(* CODESYS project CintasSoplado.project
   Title: CintasSoplado
   Version: 0.0.0.0
   Author: serbogr1

Project tree, tasks and I/O mapping:
  MyController : TM241CE40R, Schneider Electric, order no. TM241CE40R, version 4.0.6.18
    application Application
      libraries: Toolbox, 2.2.0.0 (Schneider Electric); VisuDialogs, * (System)
      task MAST (cyclic, interval 50 ms, priority 15) calls ProcesoUno, ProcesoDos, Pulsadores, PID, Gestion_HMI, Control_HMI, Soplado_AUT, Operaciones_MAT
      global variables GVL
      visualisation Control_HMIW
      image pool ImagePool
      program ProcesoDos [SFC]: E2_active, E10_active
      program PID [LD]
      program ProcesoUno [SFC]: E8_active, E7_active, E9_active, E10_active, E11_active, E12_active, E1_active
      program Pulsadores [LD]
      program Gestion_HMI [LD]
      program Control_HMI [ST]
      program Operaciones_MAT [ST]
      program Soplado_AUT [SFC]: E1_active, E3_active, E2_active, E4_active, E5_active, E6_active, E7_active
    DI : Digital Inputs, Schneider Electric, version 4.0.6.18
        input  idwDI_IDW0 : DWORD  // IDW0
        input  ibDI_IB1 : BYTE  // IB1
    DQ : Digital Outputs, Schneider Electric, version 4.0.6.18
        output qwDQ_QW0 : WORD  // QW0
        output qbDQ_QB1 : BYTE  // QB1
    Counters : Counters, Schneider Electric, version 4.0.6.18
    Pulse_Generators : Pulse Generators, Schneider Electric, version 4.0.6.18
    Cartridge_1 : Cartridge, Schneider Electric, version 4.0.6.18
      TMC4AI2 : TMC4AI2, Schneider Electric, order no. TMC4AI2, version 1.0.1.0
          input  iiTMC4AI2_IW0 : INT  // IW0
          input  iiTMC4AI2_IW1 : INT  // IW1
          input  ibTMC4AI2_IW2 : BYTE  // IW2
    Cartridge_2 : Cartridge, Schneider Electric, version 4.0.6.18
      TMC4AQ2 : TMC4AQ2, Schneider Electric, order no. TMC4AQ2, version 1.0.1.1
          output qiTMC4AQ2_QW0 : INT  // QW0
          output qiTMC4AQ2_QW1 : INT  // QW1
          input  ibTMC4AQ2_IW0 : BYTE  // IW0
    IO_Bus : IO bus - TM3, Schneider Electric, version 4.0.6.18
    COM_Bus : COM bus, Schneider Electric, version 4.0.6.18
    Ethernet_1 : Ethernet Network, Schneider Electric, version 4.0.6.18
        settings: WebServer = TRUE; FTP Server = TRUE; SoMachine Protocol = TRUE; Modbus Server = TRUE; NetManage Protocol = TRUE; SNMP protocol = TRUE; Enable Routing = FALSE; WebVisu protocol = TRUE; DHCP Server Active = FALSE
    Serial_Line_1 : Serial line, Schneider Electric, version 4.0.6.18
      SoMachine_Network_Manager : SoMachine-Network Manager, Schneider Electric, version 4.0.0.2
    Serial_Line_2 : Serial line, Schneider Electric, version 4.0.6.18
      Modbus_Manager : Modbus Manager, Schneider Electric, version 4.0.0.2
  text list GlobalTextList
*)

// MyController/Application/GVL
VAR_GLOBAL
	iTiempoFresado      AT %MW100: INT :=2;	
	iTiempoTaladrado    AT %MW101: INT :=2;
	iTiempoSoplado      AT %MW102: INT :=2;
	rReferencia         AT %MD118: REAL:=-0.75;
	iPosInicioGrados    AT %MD105: REAL:=0;
	iPosSopladoGrados   AT %MD106: REAL:=20;
    iPosSopladoReposo	AT %MD99 : REAL:=-37;
	iGradosAguja        AT %MW104: INT;
	rPosicionActual              : REAL;	
END_VAR

// MyController/Application/ProcesoUno
PROGRAM ProcesoUno
VAR
	bS_FC_Empujador_1          AT %IX0.0: BOOL; (*I1*)
	bS_IC_Empujador_1          AT %IX0.1: BOOL; (*I2*)
	bS_FC_Empujador_2          AT %IX0.2: BOOL; (*I3*)
	bS_IC_Empujador_2          AT %IX0.3: BOOL; (*I4*)
	bS_FT_Empujador_1          AT %IX0.4: BOOL; (*I5*)
	bS_FT_Fresadora            AT %IX0.5: BOOL; (*I6*)
	bS_FT_Carga                AT %IX0.6: BOOL; (*I7*)
	bS_FT_Taladro              AT %IX0.7: BOOL; (*I8*)
	bS_FT_Salida               AT %IX1.0: BOOL; (*I9*)

    bSiguientePieza            AT %MX0.4: BOOL; (*Activa cuando se puede poner la siguiente pieza*)
	FalloSensores              AT %MX0.5: BOOL:=FALSE;	
	CintaFresadoraP1                    : BOOL;	
	CintaTaladroP1                      : BOOL;	
	CintaAlimentacionP1                 : BOOL;
	MotorFresadora                      : BOOL;
END_VAR

VAR_OUTPUT
	tEmpujador_1   : TIME:=T#1S;
	tFresado       : TIME:=T#1S;
END_VAR

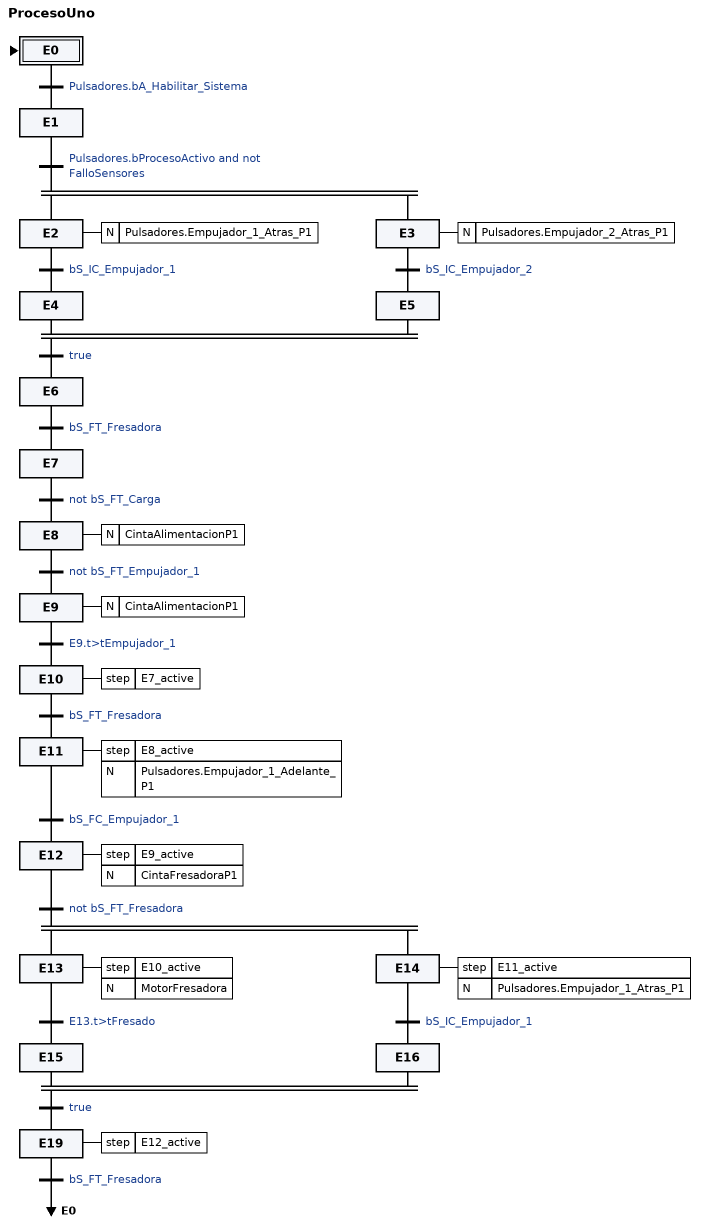
INITIAL_STEP E0:
END_STEP
TRANSITION FROM E0 TO E1
    := Pulsadores.bA_Habilitar_Sistema;
END_TRANSITION
STEP E1:
END_STEP
TRANSITION FROM E1 TO (E2, E3)
    := Pulsadores.bProcesoActivo and not FalloSensores;
END_TRANSITION
STEP E2:
    Pulsadores.Empujador_1_Atras_P1(N);
END_STEP
TRANSITION FROM E2 TO E4
    := bS_IC_Empujador_1;
END_TRANSITION
STEP E4:
END_STEP
STEP E3:
    Pulsadores.Empujador_2_Atras_P1(N);
END_STEP
TRANSITION FROM E3 TO E5
    := bS_IC_Empujador_2;
END_TRANSITION
STEP E5:
END_STEP
TRANSITION FROM (E4, E5) TO E6
    := true;
END_TRANSITION
STEP E6:
END_STEP
TRANSITION FROM E6 TO E7
    := bS_FT_Fresadora;
END_TRANSITION
STEP E7:
END_STEP
TRANSITION FROM E7 TO E8
    := not bS_FT_Carga;
END_TRANSITION
STEP E8:
    CintaAlimentacionP1(N);
END_STEP
TRANSITION FROM E8 TO E9
    := not bS_FT_Empujador_1;
END_TRANSITION
STEP E9:
    CintaAlimentacionP1(N);
END_STEP
TRANSITION FROM E9 TO E10
    := E9.t>tEmpujador_1;
END_TRANSITION
STEP E10:
    E7_active(N);  // step action
END_STEP
TRANSITION FROM E10 TO E11
    := bS_FT_Fresadora;
END_TRANSITION
STEP E11:
    E8_active(N);  // step action
    Pulsadores.Empujador_1_Adelante_P1(N);
END_STEP
TRANSITION FROM E11 TO E12
    := bS_FC_Empujador_1;
END_TRANSITION
STEP E12:
    E9_active(N);  // step action
    CintaFresadoraP1(N);
END_STEP
TRANSITION FROM E12 TO (E13, E14)
    := not bS_FT_Fresadora;
END_TRANSITION
STEP E13:
    E10_active(N);  // step action
    MotorFresadora(N);
END_STEP
TRANSITION FROM E13 TO E15
    := E13.t>tFresado;
END_TRANSITION
STEP E15:
END_STEP
STEP E14:
    E11_active(N);  // step action
    Pulsadores.Empujador_1_Atras_P1(N);
END_STEP
TRANSITION FROM E14 TO E16
    := bS_IC_Empujador_1;
END_TRANSITION
STEP E16:
END_STEP
TRANSITION FROM (E15, E16) TO E19
    := true;
END_TRANSITION
STEP E19:
    E12_active(N);  // step action
END_STEP
TRANSITION FROM E19 TO E0
    := bS_FT_Fresadora;
END_TRANSITION

ACTION E8_active:
IF bS_FT_Carga THEN
	bSiguientePieza := TRUE;
ELSIF NOT bS_FT_Carga THEN
	bSiguientePieza := FALSE;
END_IF
END_ACTION

ACTION E7_active:
IF bS_FT_Carga THEN
	bSiguientePieza := TRUE;
ELSIF NOT bS_FT_Carga THEN
	bSiguientePieza := FALSE;
END_IF
END_ACTION

ACTION E9_active:
IF bS_FT_Carga THEN
	bSiguientePieza := TRUE;
ELSIF NOT bS_FT_Carga THEN
	bSiguientePieza := FALSE;
END_IF
END_ACTION

ACTION E10_active:
IF bS_FT_Carga THEN
	bSiguientePieza := TRUE;
ELSIF NOT bS_FT_Carga THEN
	bSiguientePieza := FALSE;
END_IF

	tFresado := INT_TO_TIME(iTiempoFresado*1000);
END_ACTION

ACTION E11_active:
IF bS_FT_Carga THEN
	bSiguientePieza := TRUE;
ELSIF NOT bS_FT_Carga THEN
	bSiguientePieza := FALSE;
END_IF
END_ACTION

ACTION E12_active:
IF bS_FT_Carga THEN
	bSiguientePieza := TRUE;
ELSIF NOT bS_FT_Carga THEN
	bSiguientePieza := FALSE;
END_IF
END_ACTION

ACTION E1_active:
IF NOT Pulsadores.bBotonInicioHMIS THEN
	IF NOT bS_FT_Carga THEN
		FalloSensores:=TRUE;	
	END_IF
	IF NOT bS_FT_Empujador_1 THEN
		FalloSensores:=TRUE;
	END_IF
	IF NOT bS_FT_Fresadora THEN
		FalloSensores:=TRUE;
	END_IF
	IF NOT bS_FT_Taladro THEN
		FalloSensores:=TRUE;
	END_IF
	IF NOT bS_FT_Salida THEN
		FalloSensores:=TRUE;	
	END_IF
	
	IF bS_FT_Carga AND bS_FT_Empujador_1 AND bS_FT_Fresadora AND bS_FT_Taladro AND bS_FT_Salida THEN
		FalloSensores:=FALSE;			
	END_IF
END_IF
END_ACTION

END_PROGRAM

// MyController/Application/Pulsadores
PROGRAM Pulsadores
VAR
	bA_M_Empujador_1_Adelante  AT %QX0.4: BOOL; (*Q1*)
	bA_M_Empujador_1_Atras     AT %QX0.5: BOOL; (*Q2*)
	bA_M_Empujador_2_Adelante  AT %QX0.6: BOOL; (*Q3*)
	bA_M_Empujador_2_Atras     AT %QX0.7: BOOL; (*Q4*)	
	bA_M_Cinta_Alimentacion    AT %QX1.0: BOOL; (*Q5*)	
	bA_M_Cinta_Fresadora       AT %QX1.1: BOOL; (*Q6*)
	bA_M_Fresadora             AT %QX1.2: BOOL; (*Q7*)	
	bA_M_Cinta_Taladro         AT %QX1.3: BOOL; (*Q8*)	
	bA_M_Taladro               AT %QX1.4: BOOL; (*Q9*)	
	bA_M_Cinta_Salida          AT %QX1.5: BOOL; (*Q10*)		
	bA_Habilitar_Sistema       AT %QX1.6: BOOL; (*Q11*)	
	
	bBotonEmergenciaHMIS       AT %MX0.0: BOOL; (*Boton Emergencia HMI y HMIW*)	
	bBotonEncendidoHMIS        AT %MX0.1: BOOL; (*Boton Encendido HMI y HMIW*)	
	bBotonInicioHMIS           AT %MX0.2: BOOL; (*Boton Inicio HMI y HMIW*)	
	bAlarma_ON                 AT %MX0.3: BOOL; (*Activa cuando se pulsa alarma*)
	bProcesoActivo                      : BOOL; (*Activa cuando se pulsa inicio*)	
	
	Empujador_1_Adelante_P1             : BOOL;
	Empujador_1_Adelante_P2             : BOOL;
	Empujador_2_Adelante_P1             : BOOL;	
    Empujador_2_Adelante_P2             : BOOL;
	Empujador_1_Atras_P1                : BOOL;
	Empujador_1_Atras_P2                : BOOL;	
	Empujador_2_Atras_P1                : BOOL;
	Empujador_2_Atras_P2                : BOOL;	
	bStopSoplado                        : BOOL;	
	rLongTime                           : INT;
END_VAR

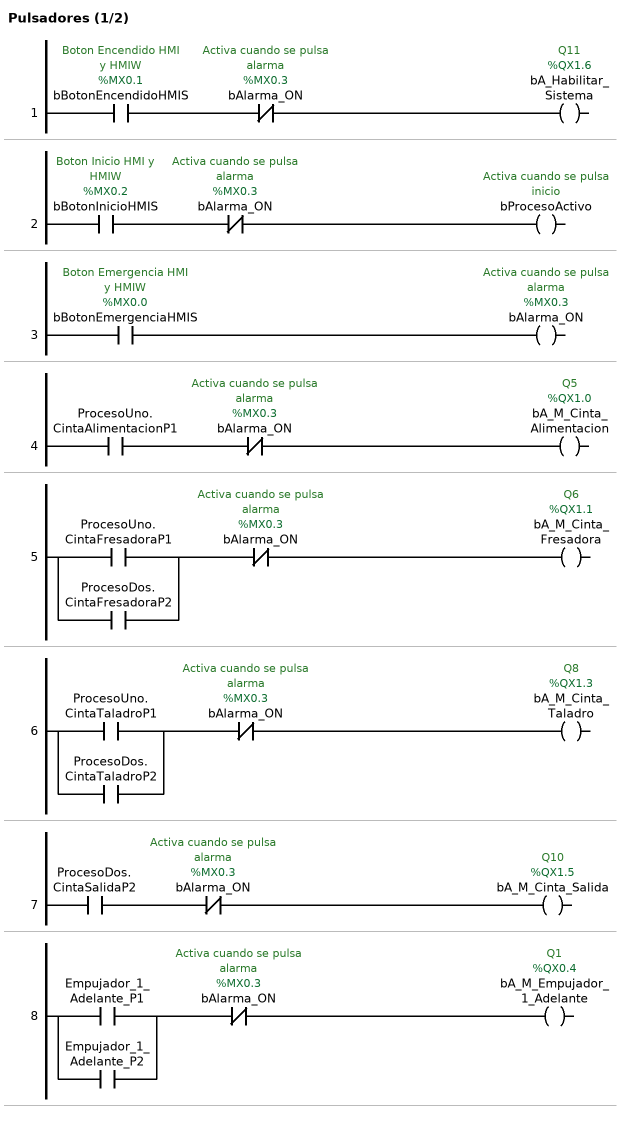
// NETWORK 1
//   bBotonEncendidoHMIS: Boton Encendido HMI y HMIW | AT %MX0.1
//   bAlarma_ON: Activa cuando se pulsa alarma | AT %MX0.3
//   bA_Habilitar_Sistema: Q11 | AT %QX1.6
bA_Habilitar_Sistema := bBotonEncendidoHMIS AND NOT bAlarma_ON;

// NETWORK 2
//   bBotonInicioHMIS: Boton Inicio HMI y HMIW | AT %MX0.2
//   bAlarma_ON: Activa cuando se pulsa alarma | AT %MX0.3
//   bProcesoActivo: Activa cuando se pulsa inicio
bProcesoActivo := bBotonInicioHMIS AND NOT bAlarma_ON;

// NETWORK 3
//   bBotonEmergenciaHMIS: Boton Emergencia HMI y HMIW | AT %MX0.0
//   bAlarma_ON: Activa cuando se pulsa alarma | AT %MX0.3
bAlarma_ON := bBotonEmergenciaHMIS;

// NETWORK 4
//   bAlarma_ON: Activa cuando se pulsa alarma | AT %MX0.3
//   bA_M_Cinta_Alimentacion: Q5 | AT %QX1.0
bA_M_Cinta_Alimentacion := ProcesoUno.CintaAlimentacionP1 AND NOT bAlarma_ON;

// NETWORK 5
//   bAlarma_ON: Activa cuando se pulsa alarma | AT %MX0.3
//   bA_M_Cinta_Fresadora: Q6 | AT %QX1.1
bA_M_Cinta_Fresadora := (ProcesoUno.CintaFresadoraP1 OR ProcesoDos.CintaFresadoraP2) AND NOT bAlarma_ON;

// NETWORK 6
//   bAlarma_ON: Activa cuando se pulsa alarma | AT %MX0.3
//   bA_M_Cinta_Taladro: Q8 | AT %QX1.3
bA_M_Cinta_Taladro := (ProcesoUno.CintaTaladroP1 OR ProcesoDos.CintaTaladroP2) AND NOT bAlarma_ON;

// NETWORK 7
//   bAlarma_ON: Activa cuando se pulsa alarma | AT %MX0.3
//   bA_M_Cinta_Salida: Q10 | AT %QX1.5
bA_M_Cinta_Salida := ProcesoDos.CintaSalidaP2 AND NOT bAlarma_ON;

// NETWORK 8
//   bAlarma_ON: Activa cuando se pulsa alarma | AT %MX0.3
//   bA_M_Empujador_1_Adelante: Q1 | AT %QX0.4
bA_M_Empujador_1_Adelante := (Empujador_1_Adelante_P1 OR Empujador_1_Adelante_P2) AND NOT bAlarma_ON;

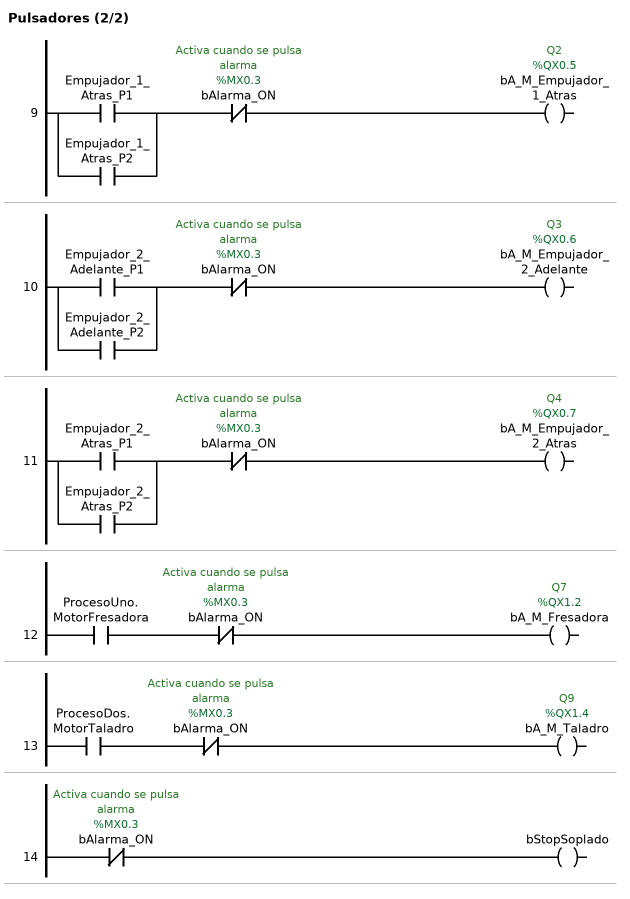
// NETWORK 9
//   bAlarma_ON: Activa cuando se pulsa alarma | AT %MX0.3
//   bA_M_Empujador_1_Atras: Q2 | AT %QX0.5
bA_M_Empujador_1_Atras := (Empujador_1_Atras_P1 OR Empujador_1_Atras_P2) AND NOT bAlarma_ON;

// NETWORK 10
//   bAlarma_ON: Activa cuando se pulsa alarma | AT %MX0.3
//   bA_M_Empujador_2_Adelante: Q3 | AT %QX0.6
bA_M_Empujador_2_Adelante := (Empujador_2_Adelante_P1 OR Empujador_2_Adelante_P2) AND NOT bAlarma_ON;

// NETWORK 11
//   bAlarma_ON: Activa cuando se pulsa alarma | AT %MX0.3
//   bA_M_Empujador_2_Atras: Q4 | AT %QX0.7
bA_M_Empujador_2_Atras := (Empujador_2_Atras_P1 OR Empujador_2_Atras_P2) AND NOT bAlarma_ON;

// NETWORK 12
//   bAlarma_ON: Activa cuando se pulsa alarma | AT %MX0.3
//   bA_M_Fresadora: Q7 | AT %QX1.2
bA_M_Fresadora := ProcesoUno.MotorFresadora AND NOT bAlarma_ON;

// NETWORK 13
//   bAlarma_ON: Activa cuando se pulsa alarma | AT %MX0.3
//   bA_M_Taladro: Q9 | AT %QX1.4
bA_M_Taladro := ProcesoDos.MotorTaladro AND NOT bAlarma_ON;

// NETWORK 14
//   bAlarma_ON: Activa cuando se pulsa alarma | AT %MX0.3
bStopSoplado := NOT bAlarma_ON;

END_PROGRAM

// MyController/Application/ProcesoDos
PROGRAM ProcesoDos
VAR	
    CintaSalidaP2                 : BOOL;
    MotorTaladro                  : BOOL;
	CintaFresadoraP2              : BOOL;
	CintaTaladroP2                : BOOL;	

	rPiezasTerminadas   AT %MW103 : INT:=0;		
	tTaladrado                    : TIME:=T#2S;
	tEmpujador_2                  : TIME:=T#2S;	
END_VAR

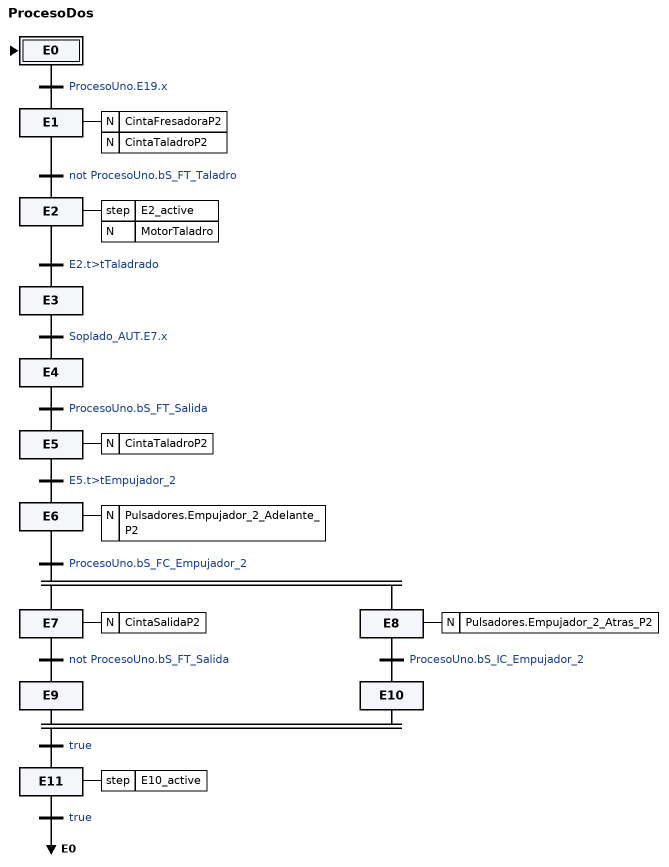
INITIAL_STEP E0:
END_STEP
TRANSITION FROM E0 TO E1
    := ProcesoUno.E19.x;
END_TRANSITION
STEP E1:
    CintaFresadoraP2(N);
    CintaTaladroP2(N);
END_STEP
TRANSITION FROM E1 TO E2
    := not ProcesoUno.bS_FT_Taladro;
END_TRANSITION
STEP E2:
    E2_active(N);  // step action
    MotorTaladro(N);
END_STEP
TRANSITION FROM E2 TO E3
    := E2.t>tTaladrado;
END_TRANSITION
STEP E3:
END_STEP
TRANSITION FROM E3 TO E4
    := Soplado_AUT.E7.x;
END_TRANSITION
STEP E4:
END_STEP
TRANSITION FROM E4 TO E5
    := ProcesoUno.bS_FT_Salida;
END_TRANSITION
STEP E5:
    CintaTaladroP2(N);
END_STEP
TRANSITION FROM E5 TO E6
    := E5.t>tEmpujador_2;
END_TRANSITION
STEP E6:
    Pulsadores.Empujador_2_Adelante_P2(N);
END_STEP
TRANSITION FROM E6 TO (E7, E8)
    := ProcesoUno.bS_FC_Empujador_2;
END_TRANSITION
STEP E7:
    CintaSalidaP2(N);
END_STEP
TRANSITION FROM E7 TO E9
    := not ProcesoUno.bS_FT_Salida;
END_TRANSITION
STEP E9:
END_STEP
STEP E8:
    Pulsadores.Empujador_2_Atras_P2(N);
END_STEP
TRANSITION FROM E8 TO E10
    := ProcesoUno.bS_IC_Empujador_2;
END_TRANSITION
STEP E10:
END_STEP
TRANSITION FROM (E9, E10) TO E11
    := true;
END_TRANSITION
STEP E11:
    E10_active(N);  // step action
END_STEP
TRANSITION FROM E11 TO E0
    := true;
END_TRANSITION

ACTION E2_active:
  
IF Gestion_HMI.bSum_T_Taladrado THEN
	iTiempoTaladrado := iTiempoTaladrado + 1;
END_IF
IF Gestion_HMI.bRes_T_Taladrado THEN
	iTiempoTaladrado := iTiempoTaladrado - 1;
END_IF

	tTaladrado := INT_TO_TIME(iTiempoTaladrado*1000);
END_ACTION

ACTION E10_active:
IF NOT ProcesoUno.bS_FT_Salida THEN
	rPiezasTerminadas := rPiezasTerminadas + 1;
END_IF
END_ACTION

END_PROGRAM

// MyController/Application/Gestion_HMI
PROGRAM Gestion_HMI
VAR
	bRes_T_Fresado              AT %MX1.0: BOOL;
	bSum_T_Fresado              AT %MX1.1: BOOL;
	bRes_T_Taladrado            AT %MX1.2: BOOL;
	bSum_T_Taladrado            AT %MX1.3: BOOL;
	bRes_T_Soplado              AT %MX1.4: BOOL;
	bSum_T_Soplado              AT %MX1.5: BOOL;		
	bRes_AnguloInicio           AT %MX1.6: BOOL;		
	bSum_AnguloInicio           AT %MX1.7: BOOL;
	bRes_AnguloSoplado          AT %MX2.0: BOOL;
	bSum_AnguloSoplado          AT %MX2.1: BOOL;	

	bSe_FT_Carga                AT %MX2.2: BOOL; 
	bSe_FT_Empujador_1          AT %MX2.3: BOOL; 
	bSe_FC_Empujador_1          AT %MX2.4: BOOL;
	bSe_FT_Fresadora            AT %MX2.5: BOOL; 	
	bSe_FT_Taladro              AT %MX2.6: BOOL;
	bSe_FC_Empujador_2          AT %MX2.7: BOOL;  
	bSe_FT_Salida               AT %MX3.0: BOOL; 
	bAe_M_Empujador_1_Adelante  AT %MX3.1: BOOL;
	bAe_M_Fresadora             AT %MX3.2: BOOL;
	bAe_M_Taladro               AT %MX3.3: BOOL;
	bAe_M_Empujador_2_Adelante  AT %MX3.4: BOOL;	

END_VAR

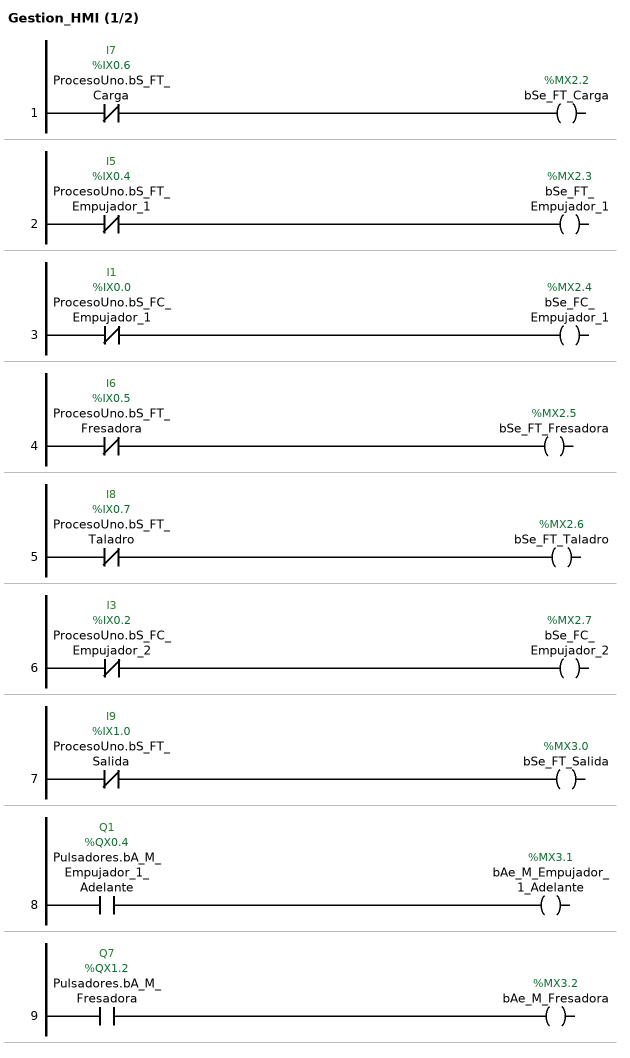
// NETWORK 1
//   ProcesoUno.bS_FT_Carga: I7 | AT %IX0.6
//   bSe_FT_Carga: AT %MX2.2
bSe_FT_Carga := NOT ProcesoUno.bS_FT_Carga;

// NETWORK 2
//   ProcesoUno.bS_FT_Empujador_1: I5 | AT %IX0.4
//   bSe_FT_Empujador_1: AT %MX2.3
bSe_FT_Empujador_1 := NOT ProcesoUno.bS_FT_Empujador_1;

// NETWORK 3
//   ProcesoUno.bS_FC_Empujador_1: I1 | AT %IX0.0
//   bSe_FC_Empujador_1: AT %MX2.4
bSe_FC_Empujador_1 := NOT ProcesoUno.bS_FC_Empujador_1;

// NETWORK 4
//   ProcesoUno.bS_FT_Fresadora: I6 | AT %IX0.5
//   bSe_FT_Fresadora: AT %MX2.5
bSe_FT_Fresadora := NOT ProcesoUno.bS_FT_Fresadora;

// NETWORK 5
//   ProcesoUno.bS_FT_Taladro: I8 | AT %IX0.7
//   bSe_FT_Taladro: AT %MX2.6
bSe_FT_Taladro := NOT ProcesoUno.bS_FT_Taladro;

// NETWORK 6
//   ProcesoUno.bS_FC_Empujador_2: I3 | AT %IX0.2
//   bSe_FC_Empujador_2: AT %MX2.7
bSe_FC_Empujador_2 := NOT ProcesoUno.bS_FC_Empujador_2;

// NETWORK 7
//   ProcesoUno.bS_FT_Salida: I9 | AT %IX1.0
//   bSe_FT_Salida: AT %MX3.0
bSe_FT_Salida := NOT ProcesoUno.bS_FT_Salida;

// NETWORK 8
//   Pulsadores.bA_M_Empujador_1_Adelante: Q1 | AT %QX0.4
//   bAe_M_Empujador_1_Adelante: AT %MX3.1
bAe_M_Empujador_1_Adelante := Pulsadores.bA_M_Empujador_1_Adelante;

// NETWORK 9
//   Pulsadores.bA_M_Fresadora: Q7 | AT %QX1.2
//   bAe_M_Fresadora: AT %MX3.2
bAe_M_Fresadora := Pulsadores.bA_M_Fresadora;

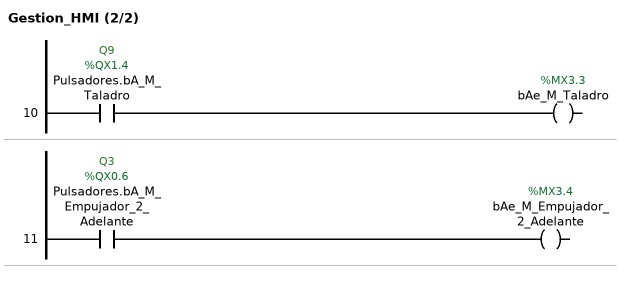
// NETWORK 10
//   Pulsadores.bA_M_Taladro: Q9 | AT %QX1.4
//   bAe_M_Taladro: AT %MX3.3
bAe_M_Taladro := Pulsadores.bA_M_Taladro;

// NETWORK 11
//   Pulsadores.bA_M_Empujador_2_Adelante: Q3 | AT %QX0.6
//   bAe_M_Empujador_2_Adelante: AT %MX3.4
bAe_M_Empujador_2_Adelante := Pulsadores.bA_M_Empujador_2_Adelante;

END_PROGRAM

// MyController/Application/PID
PROGRAM PID
VAR
	vActuador              AT %QW2   : WORD;
	vSensor                AT %IW3   : WORD;
	vSensorSimu                      : WORD:=2500;	
	vActuador_PID          AT %MW110 : WORD;
	vSensor_PID            AT %MW111 : WORD;	
	rActuador              AT %MD114 : REAL:=0;
	rSensor                          : REAL:=0;	
	rOutPIDgrados                    : REAL;
	rV_Equilibrio                    : REAL:=3.85509;

	bBotonAutMan_PID       AT %MX0.06: BOOL;
	bBotonReset_PID        AT %MX0.07: BOOL;	

	rKp                    AT %MD115 : REAL:=0.2008;
	rKi                    AT %MD116 : REAL:=0.1358;
	rKd                    AT %MD117 : REAL:=1.2154;
	
	wKp                    AT %MW90  : WORD;
	wKi                    AT %MW91  : WORD;
	wKd                    AT %MW92  : WORD;

	FB_Scaling_vS                    : FB_Scaling; (*Escalado para tensión del sensor*)
	FB_Scaling_vA                    : FB_Scaling; (*Escalado para tensión al actuador*)
	PID_ControHelice                 : Util.PID;
	
END_VAR
VAR // added by the converter: edge detectors and wires of the graphical bodies
    _w1 : BOOL;
END_VAR

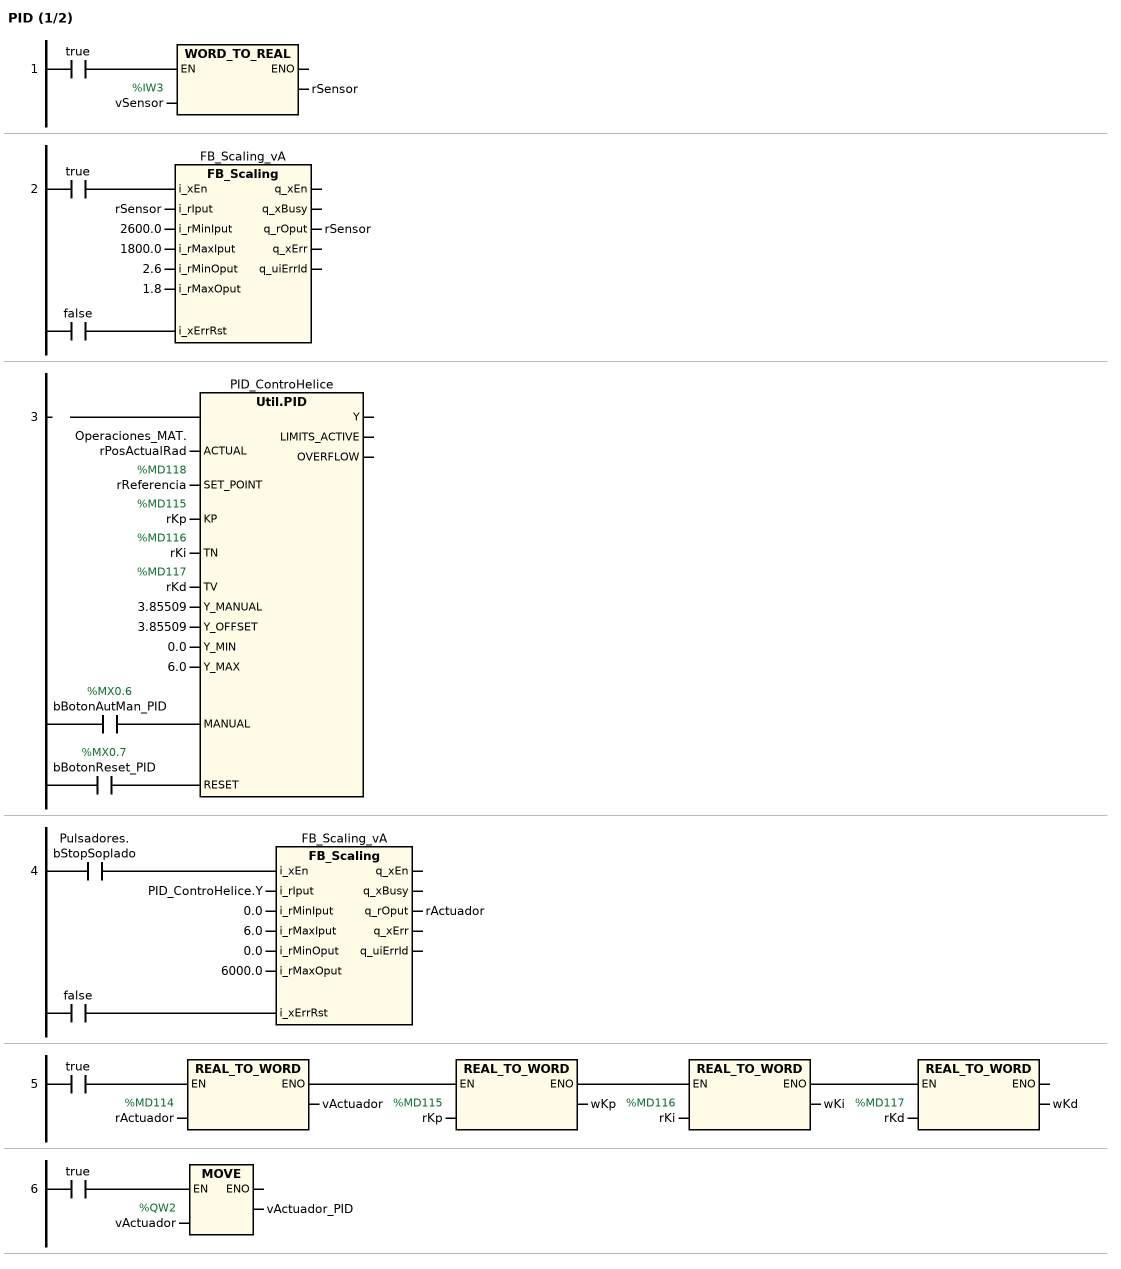
// NETWORK 1
//   vSensor: AT %IW3
IF true THEN rSensor := WORD_TO_REAL(vSensor); END_IF

// NETWORK 2
//   FB_Scaling_vA: Escalado para tensión al actuador
FB_Scaling_vA(
    i_xEn := true,
    i_rIput := rSensor,
    i_rMinIput := 2600.0,
    i_rMaxIput := 1800.0,
    i_rMinOput := 2.6,
    i_rMaxOput := 1.8,
    i_xErrRst := false,
    q_rOput => rSensor); // FB_Scaling

// NETWORK 3
//   rReferencia: AT %MD118
//   rKp: AT %MD115
//   rKi: AT %MD116
//   rKd: AT %MD117
//   bBotonAutMan_PID: AT %MX0.6
//   bBotonReset_PID: AT %MX0.7
PID_ControHelice(
    ACTUAL := Operaciones_MAT.rPosActualRad,
    SET_POINT := rReferencia,
    KP := rKp,
    TN := rKi,
    TV := rKd,
    Y_MANUAL := 3.85509,
    Y_OFFSET := 3.85509,
    Y_MIN := 0.0,
    Y_MAX := 6.0,
    MANUAL := bBotonAutMan_PID,
    RESET := bBotonReset_PID); // Util.PID

// NETWORK 4
//   FB_Scaling_vA: Escalado para tensión al actuador
//   PID_ControHelice.Y: manipulated variable, set value
//   rActuador: AT %MD114
FB_Scaling_vA(
    i_xEn := Pulsadores.bStopSoplado,
    i_rIput := PID_ControHelice.Y,
    i_rMinIput := 0.0,
    i_rMaxIput := 6.0,
    i_rMinOput := 0.0,
    i_rMaxOput := 6000.0,
    i_xErrRst := false,
    q_rOput => rActuador); // FB_Scaling

// NETWORK 5
//   rActuador: AT %MD114
//   vActuador: AT %QW2
//   rKp: AT %MD115
//   wKp: AT %MW90
//   rKi: AT %MD116
//   wKi: AT %MW91
//   rKd: AT %MD117
//   wKd: AT %MW92
_w1 := true;
IF _w1 THEN vActuador := REAL_TO_WORD(rActuador); END_IF
IF _w1 THEN wKp := REAL_TO_WORD(rKp); END_IF
IF _w1 THEN wKi := REAL_TO_WORD(rKi); END_IF
IF _w1 THEN wKd := REAL_TO_WORD(rKd); END_IF

// NETWORK 6
//   vActuador: AT %QW2
//   vActuador_PID: AT %MW110
IF true THEN vActuador_PID := vActuador; END_IF

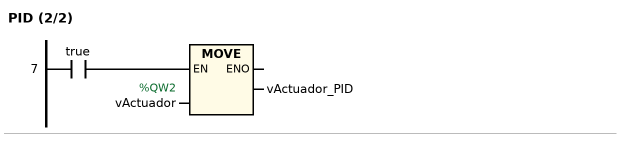
// NETWORK 7
//   vActuador: AT %QW2
//   vActuador_PID: AT %MW110
IF true THEN vActuador_PID := vActuador; END_IF

END_PROGRAM

// MyController/Application/Operaciones_MAT
PROGRAM Operaciones_MAT
VAR
	rActuador                      : REAL:=0;
	iPosReposo                     : INT:=0;
	iPosInicio           AT %MD112 : REAL:=0;
	iPosSoplado          AT %MD113 : REAL:=0;		
    step                           : INT:=1;	
	tTiempoSoplado                 : TIME:=T#2S;
	rPosActualRad: LREAL;
	wReferencia          At %MW119 : WORD;
END_VAR


rPosicionActual := -81.93 * PID.rSensor + 178.42;

rPosActualRad := (rPosicionActual * 3.1415)/180;

iGradosAguja := REAL_TO_INT(rPosicionActual);

(*iGradosAguja := REAL_TO_INT((PID.PID_ControHelice.Y - 2.7533) / 0.0833);*)

tTiempoSoplado := INT_TO_TIME(iTiempoSoplado*1000);

wReferencia := REAL_TO_WORD(rReferencia);

END_PROGRAM

// MyController/Application/Control_HMI
PROGRAM Control_HMI
VAR
END_VAR



IF Gestion_HMI.bSum_T_Fresado THEN              (*Incremento/decremento desde HMI el tiempo de fresado*)
	iTiempoFresado := iTiempoFresado + 1;
	
END_IF
IF Gestion_HMI.bRes_T_Fresado THEN
	iTiempoFresado := iTiempoFresado - 1;
END_IF

IF Gestion_HMI.bSum_T_Taladrado THEN              (*Incremento/decremento desde HMI el tiempo de taladrado*)
	iTiempoTaladrado := iTiempoTaladrado + 1;
	
END_IF
IF Gestion_HMI.bRes_T_Taladrado THEN
	iTiempoTaladrado := iTiempoTaladrado - 1;
END_IF

IF Gestion_HMI.bSum_T_Soplado THEN              (*Incremento/dexcremento desde HMI el tiempo de soplado*)
	iTiempoSoplado := iTiempoSoplado + 1;
	
END_IF
IF Gestion_HMI.bRes_T_Soplado THEN
	iTiempoSoplado := iTiempoSoplado - 1;
END_IF

IF Gestion_HMI.bSum_AnguloInicio THEN           (*Incremento/dexcremento desde HMI el angulo de inicio*)
	iPosInicioGrados := iPosInicioGrados + 1;
END_IF
IF Gestion_HMI.bRes_AnguloInicio THEN
	iPosInicioGrados := iPosInicioGrados - 1;
END_IF

IF Gestion_HMI.bSum_AnguloSoplado THEN           (*Incremento/dexcremento desde HMI el angulo de soplado*)
	iPosSopladoGrados := iPosSopladoGrados + 1;
END_IF
IF Gestion_HMI.bRes_AnguloSoplado THEN
	iPosSopladoGrados := iPosSopladoGrados - 1;
END_IF

END_PROGRAM

// MyController/Application/Soplado_AUT
PROGRAM Soplado_AUT
VAR
	bReferenciaAlcanzada     : BOOL:=FALSE;
	bFinSoplado_AUT          : BOOL:=FALSE;
END_VAR

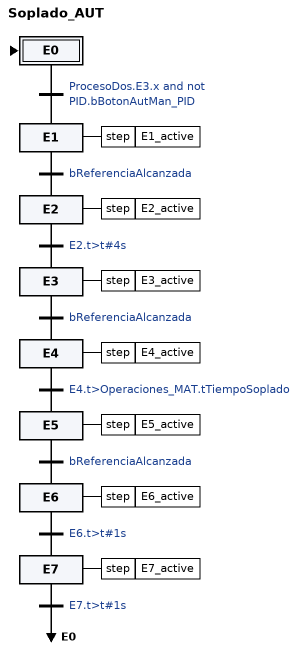
INITIAL_STEP E0:
END_STEP
TRANSITION FROM E0 TO E1
    := ProcesoDos.E3.x and not PID.bBotonAutMan_PID;
END_TRANSITION
STEP E1:
    E1_active(N);  // step action
END_STEP
TRANSITION FROM E1 TO E2
    := bReferenciaAlcanzada;
END_TRANSITION
STEP E2:
    E2_active(N);  // step action
END_STEP
TRANSITION FROM E2 TO E3
    := E2.t>t#4s;
END_TRANSITION
STEP E3:
    E3_active(N);  // step action
END_STEP
TRANSITION FROM E3 TO E4
    := bReferenciaAlcanzada;
END_TRANSITION
STEP E4:
    E4_active(N);  // step action
END_STEP
TRANSITION FROM E4 TO E5
    := E4.t>Operaciones_MAT.tTiempoSoplado;
END_TRANSITION
STEP E5:
    E5_active(N);  // step action
END_STEP
TRANSITION FROM E5 TO E6
    := bReferenciaAlcanzada;
END_TRANSITION
STEP E6:
    E6_active(N);  // step action
END_STEP
TRANSITION FROM E6 TO E7
    := E6.t>t#1s;
END_TRANSITION
STEP E7:
    E7_active(N);  // step action
END_STEP
TRANSITION FROM E7 TO E0
    := E7.t>t#1s;
END_TRANSITION

ACTION E1_active:

	rReferencia := (iPosInicioGrados*3.1415)/180;
	
	IF PID.vActuador >= PID.rV_Equilibrio THEN
		bReferenciaAlcanzada:=TRUE;
	END_IF
END_ACTION

ACTION E3_active:

	rReferencia := (iPosSopladoGrados*3.1415)/180;
	
	IF PID.vActuador >= 5000 THEN
		bReferenciaAlcanzada:=TRUE;
	END_IF
END_ACTION

ACTION E2_active:

	bReferenciaAlcanzada := FALSE;
END_ACTION

ACTION E4_active:

	bReferenciaAlcanzada:=FALSE;
END_ACTION

ACTION E5_active:

	rReferencia := (iPosInicioGrados * 3.1415)/180;
	
	IF PID.vActuador <= 3900 THEN
		bReferenciaAlcanzada:=TRUE;
	END_IF
END_ACTION

ACTION E6_active:

	rReferencia := (iPosSopladoReposo * 3.1415)/180;
	
	IF PID.vActuador <= 500 THEN
		bReferenciaAlcanzada:=TRUE;
	END_IF
END_ACTION

ACTION E7_active:
	bReferenciaAlcanzada:=FALSE;
END_ACTION

END_PROGRAM

// MyController/Application/Control_HMIW
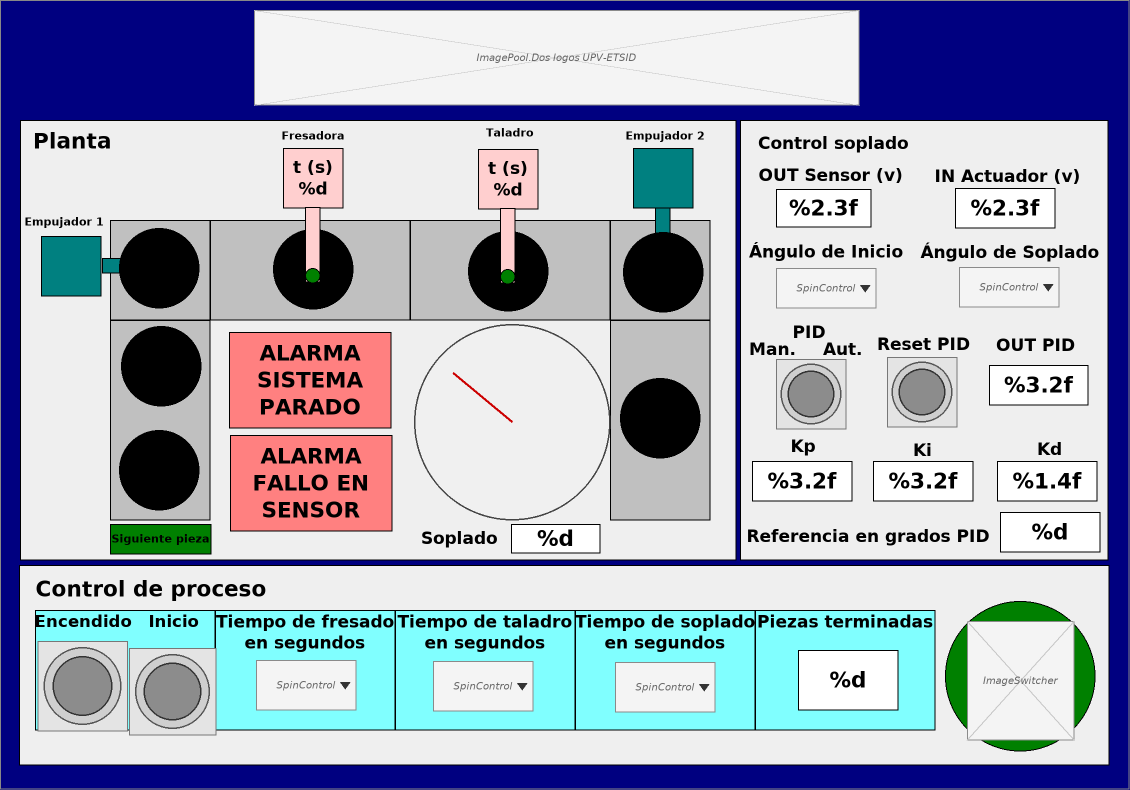
VISUALIZATION Control_HMIW  // 1130x790
    Rectangle (740,120 368x440)
    Rectangle (20,120 716x440)
    Rectangle (19,565 1090x200)
    Rectangle (110,220 100x100)
    Rectangle (110,320 100x200)
    Rectangle (610,320 100x200)
    Rectangle (610,220 100x100)
    Rectangle (210,220 200x100)
    Rectangle (410,220 200x100)
    Rectangle (35,610 180x120), "Encendido Inicio"
    Rectangle (215,610 180x120), "Tiempo de fresado en segundos"
    Rectangle (395,610 180x120), "Tiempo de taladro en segundos"
    Rectangle (575,610 180x120), "Tiempo de soplado en segundos"
    Rectangle (755,610 180x120), "Piezas terminadas"
    Label (40,574 222x30), "Control de proceso"
    SpinControl (256,660 100x50), variable: iTiempoFresado
    PushSwitchLed (37,641 91x90), variable: Pulsadores.bBotonEncendidoHMIS, behaviour: TOGGLE, style: Switch-PushSwitchLed-Gray
    Ellipse (119,430 80x80), invisible if: ProcesoUno.bS_FT_Carga
    Ellipse (121,326 80x80), invisible if: ProcesoUno.bS_FT_Empujador_1
    Ellipse (273,229 80x80), invisible if: ProcesoUno.bS_FT_Fresadora
    Ellipse (468,231 80x80), invisible if: ProcesoUno.bS_FT_Taladro
    Ellipse (620,378 80x80), invisible if: ProcesoUno.bS_FT_Salida
    RoundedRectangle (798,650 100x60), "%d", text variable: ProcesoDos.rPiezasTerminadas
    RoundedRectangle (41,236 60x60)
    RoundedRectangle (283,148 60x60), "t (s) %d", text variable: ProcesoUno.E13.t/1000, colour toggle: ProcesoUno.MotorFresadora
    RoundedRectangle (478,149 60x60), "t (s) %d", text variable: ProcesoDos.E2.t/1000, colour toggle: ProcesoDos.MotorTaladro
    Rectangle (305,207 15x75), colour toggle: ProcesoUno.MotorFresadora
    Rectangle (500,208 15x75), colour toggle: ProcesoDos.MotorTaladro
    Rectangle (655,205 15x75), invisible if: not Pulsadores.bA_M_Empujador_2_Adelante
    Ellipse (305,268 15x15), colour toggle: ProcesoUno.MotorFresadora
    Ellipse (500,269 15x15), colour toggle: ProcesoDos.MotorTaladro
    Rectangle (102,258 75x15), invisible if: not Pulsadores.bA_M_Empujador_1_Adelante
    Ellipse (623,232 80x80), invisible if: ProcesoUno.bS_IC_Empujador_2
    Label (277,121 72x30), "Fresadora"
    Label (23,207 82x30), "Empujador 1"
    Label (475,118 70x30), "Taladro"
    Label (629,121 72x30), "Empujador 2"
    Image (254,10 605x95), image: ImagePool.Dos logos UPV-ETSID
    Label (27,127 91x28), "Planta"
    Ellipse (945,601 150x150), colour toggle: Pulsadores.bBotonEmergenciaHMIS
    ImageSwitcher (967,621 107x119), variable: Pulsadores.bBotonEmergenciaHMIS, background image: ImagePool.BotonEmergencia, image: ImagePool.BotonEmergencia, behaviour: TOGGLE
    RoundedRectangle (110,524 101x30), "Siguiente pieza", colour toggle: ProcesoUno.bSiguientePieza
    Label (757,160 148x30), "OUT Sensor (v)"
    Label (747,521 242x30), "Referencia en grados PID"
    Label (934,161 147x30), "IN Actuador (v)"
    Label (972,330 127x30), "OUT PID"
    RoundedRectangle (776,189 95x38), "%2.3f", text variable: PID.rSensor
    RoundedRectangle (955,188 100x40), "%2.3f", text variable: PID.rActuador/1000
    RoundedRectangle (1000,512 100x40), "%d", text variable: rReferencia
    Label (751,128 165x30), "Control soplado"
    PushSwitchLed (129,641 87x101), variable: Pulsadores.bBotonInicioHMIS, behaviour: TAP, style: Switch-PushSwitchLed-Gray
    Meter90 (413,324 198x196), value: iGradosAguja, style: Meter-Meter90-Gray, scale format: %d, scale -40..40
    RoundedRectangle (989,365 99x40), "%3.2f", text variable: PID.PID_ControHelice.Y
    SpinControl (776,268 100x40), variable: iPosInicioGrados
    SpinControl (959,267 100x40), variable: iPosSopladoGrados
    Label (753,237 152x29), "Ángulo de Inicio"
    Label (920,237 180x30), "Ángulo de Soplado"
    RoundedRectangle (229,332 162x96), "ALARMA SISTEMA PARADO", invisible if: not Pulsadores.bAlarma_ON
    RoundedRectangle (230,435 162x96), "ALARMA FALLO EN SENSOR", invisible if: not ProcesoUno.FalloSensores
    Ellipse (119,228 80x80), invisible if: ProcesoUno.bS_IC_Empujador_1
    PushSwitch (887,357 70x70), variable: PID.bBotonReset_PID, behaviour: TAP, style: Switch-PushSwitch-Gray
    Label (860,329 127x30), "Reset PID"
    Label (787,317 44x30), "PID"
    PushSwitchLed (776,359 70x70), variable: PID.bBotonAutMan_PID, behaviour: TOGGLE, style: Switch-PushSwitchLed-Gray
    Label (385,523 149x30), "Soplado"
    RoundedRectangle (633,148 60x60)
    SpinControl (433,661 100x50), variable: iTiempoTaladrado
    SpinControl (615,662 100x50), variable: iTiempoSoplado
    RoundedRectangle (752,461 100x40), "%3.2f", text variable: PID.rKp
        OnMouseDown: write the text variable via VisuDialogs.Numpad, min -100, max 500
    RoundedRectangle (873,461 100x40), "%3.2f", text variable: PID.rKi
        OnMouseDown: write the text variable via VisuDialogs.Numpad, min -100, max 500
    RoundedRectangle (997,461 100x40), "%1.4f", text variable: PID.rKd
        OnMouseDown: write the text variable via VisuDialogs.Numpad, min -100, max 500
    Label (758,431 90x30), "Kp"
    Label (878,435 89x30), "Ki"
    Label (1002,434 95x30), "Kd"
    Label (751,334 43x30), "Man."
    Label (818,334 50x30), "Aut."
    RoundedRectangle (511,524 89x29), "%d", text variable: iGradosAguja
END_VISUALIZATION
